// Shift data from end to begin
FUNCTION ShiftDataRight : BOOL
VAR_INPUT
	data : ANY;
	byteCount : UDINT; // How far to the right are shifted
END_VAR

MEMMOVE(destAddr := data.pValue + byteCount, srcAddr := data.pValue, n := TO_UDINT(data.diSize) - byteCount);
MEMSET(destAddr := data.pValue, fillByte := 0, n := byteCount);

END_FUNCTION

(* stored: Version 1.1.0.1
   POU ShiftDataRight: Id {2f7c7bf6-f211-0025-110b-2dcfdf5fefc4}, SpecialFunc None *)
